PROGRAM MAIN
VAR
END_VAR

END_PROGRAM

(* stored: Version 1.1.0.1
   POU MAIN: Id {7b316274-9c8c-43fa-ac00-fbcea73629c0} *)
